// TIA Portal V18 export
// export: Created 2026-06-08T16:32:20.2868061Z, ExportSetting WithDefaults, DisplayName Totally Integrated Automation Portal, DisplayVersion V18, DisplayName TIA Portal Openness, DisplayVersion V18, DisplayName TIA Portal Version Control Interface, DisplayVersion V18, DisplayName STEP 7 Professional, DisplayVersion V18, DisplayName STEP 7 Safety, DisplayVersion V18, DisplayName WinCC Professional, DisplayVersion V18
FUNCTION_BLOCK "PICK_UP_LID_ROBOT"   // FB1, LAD
VERSION : 0.1
// stored: AutoNumber true, IsIECCheckEnabled false, UDAEnableTagReadback false
   VAR_TEMP   // added for the SCL form of the ladder/FBD networks
      _w1 : Bool;
   END_VAR
BEGIN

REGION Network 1: LID_PICKUP_ROBOT_LOWERING_Z_AXIS
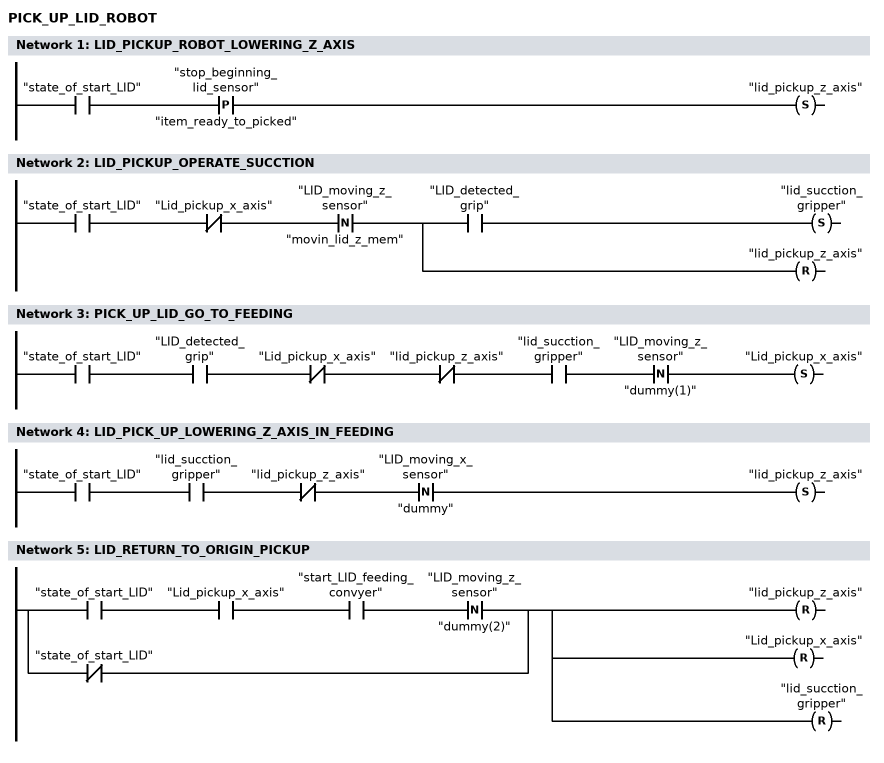
   RUNG wire#powerrail
      Contact( "state_of_start_LID" )
      P_Contact(operand := "stop_beginning_lid_sensor", bit := "item_ready_to_picked")
      S_Coil( "lid_pickup_z_axis" )
   END_RUNG
   // the same network as SCL:
   #_w1 := "state_of_start_LID" AND "stop_beginning_lid_sensor" AND NOT "item_ready_to_picked";   // rising edge of "stop_beginning_lid_sensor"
   "item_ready_to_picked" := "stop_beginning_lid_sensor";
   IF #_w1 THEN "lid_pickup_z_axis" := TRUE; END_IF;
END_REGION

REGION Network 2: LID_PICKUP_OPERATE_SUCCTION
   RUNG wire#powerrail
      Contact( "state_of_start_LID" )
      I_Contact( "Lid_pickup_x_axis" )
      N_Contact(operand := "LID_moving_z_sensor", bit := "movin_lid_z_mem")
      wire#w1
      Contact( "LID_detected_grip" )
      S_Coil( "lid_sucction_gripper" )
   END_RUNG
   RUNG wire#w1
      R_Coil( "lid_pickup_z_axis" )
   END_RUNG
   // the same network as SCL:
   #_w1 := "state_of_start_LID" AND NOT "Lid_pickup_x_axis" AND NOT "LID_moving_z_sensor" AND "movin_lid_z_mem";   // falling edge of "LID_moving_z_sensor"
   "movin_lid_z_mem" := "LID_moving_z_sensor";
   IF #_w1 AND "LID_detected_grip" THEN "lid_sucction_gripper" := TRUE; END_IF;
   IF #_w1 THEN "lid_pickup_z_axis" := FALSE; END_IF;
END_REGION

REGION Network 3: PICK_UP_LID_GO_TO_FEEDING
   RUNG wire#powerrail
      Contact( "state_of_start_LID" )
      Contact( "LID_detected_grip" )
      I_Contact( "Lid_pickup_x_axis" )
      I_Contact( "lid_pickup_z_axis" )
      Contact( "lid_sucction_gripper" )
      N_Contact(operand := "LID_moving_z_sensor", bit := "dummy(1)")
      S_Coil( "Lid_pickup_x_axis" )
   END_RUNG
   // the same network as SCL:
   #_w1 := "state_of_start_LID" AND "LID_detected_grip" AND NOT "Lid_pickup_x_axis" AND NOT "lid_pickup_z_axis" AND "lid_sucction_gripper" AND NOT "LID_moving_z_sensor" AND "dummy(1)";   // falling edge of "LID_moving_z_sensor"
   "dummy(1)" := "LID_moving_z_sensor";
   IF #_w1 THEN "Lid_pickup_x_axis" := TRUE; END_IF;
END_REGION

REGION Network 4: LID_PICK_UP_LOWERING_Z_AXIS_IN_FEEDING
   RUNG wire#powerrail
      Contact( "state_of_start_LID" )
      Contact( "lid_sucction_gripper" )
      I_Contact( "lid_pickup_z_axis" )
      N_Contact(operand := "LID_moving_x_sensor", bit := "dummy")
      S_Coil( "lid_pickup_z_axis" )
   END_RUNG
   // the same network as SCL:
   #_w1 := "state_of_start_LID" AND "lid_sucction_gripper" AND NOT "lid_pickup_z_axis" AND NOT "LID_moving_x_sensor" AND "dummy";   // falling edge of "LID_moving_x_sensor"
   "dummy" := "LID_moving_x_sensor";
   IF #_w1 THEN "lid_pickup_z_axis" := TRUE; END_IF;
END_REGION

REGION Network 5: LID_RETURN_TO_ORIGIN_PICKUP
   RUNG wire#powerrail
      Contact( "state_of_start_LID" )
      Contact( "Lid_pickup_x_axis" )
      Contact( "start_LID_feeding_convyer" )
      N_Contact(operand := "LID_moving_z_sensor", bit := "dummy(2)")
      wire#w1
      R_Coil( "lid_pickup_z_axis" )
   END_RUNG
   RUNG wire#powerrail
      I_Contact( "state_of_start_LID" )
   END_RUNG wire#w1
   RUNG wire#w1
      R_Coil( "Lid_pickup_x_axis" )
   END_RUNG
   RUNG wire#w1
      R_Coil( "lid_sucction_gripper" )
   END_RUNG
   // the same network as SCL:
   #_w1 := "state_of_start_LID" AND "Lid_pickup_x_axis" AND "start_LID_feeding_convyer" AND NOT "LID_moving_z_sensor" AND "dummy(2)";   // falling edge of "LID_moving_z_sensor"
   "dummy(2)" := "LID_moving_z_sensor";
   IF #_w1 OR NOT "state_of_start_LID" THEN
       "lid_pickup_z_axis" := FALSE;
       "Lid_pickup_x_axis" := FALSE;
       "lid_sucction_gripper" := FALSE;
   END_IF;
END_REGION
END_FUNCTION_BLOCK
